// TwinCAT 3 PLC project PLC
// ProgramVersion: 3.1.4024.0
// libraries:
//   Tc2_Standard, * (Beckhoff Automation GmbH)
//   Tc2_System, * (Beckhoff Automation GmbH)
//   Tc3_Module, * (Beckhoff Automation GmbH)
//   VisuDialogs, * (System)
//   VisuSymbols,3.5.10.0,System
// project tree:
//   / GlobalTextList.TcGTLO (not stored), PlcTask.TcTTO, Visualization Manager.TcVMO (not stored)
//   POUs/ MAIN.TcPOU
//   VISUs/ Visualization.TcVIS
// real-time tasks:
//   TASK PlcTask: cycle T#10ms, priority 20, ADS port 350

CONFIGURATION PLC
    RESOURCE PLC ON TwinCAT3
        TASK PlcTask(INTERVAL := T#10ms, PRIORITY := 20);
        PROGRAM MAIN WITH PlcTask : MAIN;
    END_RESOURCE
END_CONFIGURATION

// ---- POUs/MAIN.TcPOU
PROGRAM MAIN
VAR
	bStartMotor : BOOL := FALSE;
	bStopMotor  : BOOL := FALSE;
	bServoMotor : BOOL;
	sr_MotorSetReset : SR;
END_VAR


sr_MotorSetReset(SET1:= bStartMotor,
				 RESET:= bStopMotor,
				 Q1 => bServoMotor);

END_PROGRAM

// ---- VISUs/Visualization.TcVIS
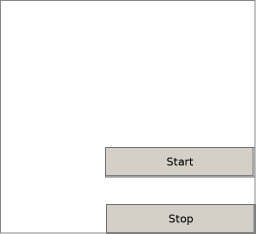
VISUALIZATION Visualization  // 256x234
    Button (105,147 150x30), "Start"
        OnMouseDown: execute { MAIN.bStartMotor := TRUE; }
        OnMouseUp: execute { MAIN.bStartMotor :=  FALSE; }
    Button (106,204 150x30), "Stop", pressed state: MAIN.bStopMotor
        OnMouseDown: execute { MAIN.bStopMotor := TRUE; }
        OnMouseUp: execute { MAIN.bStopMotor := FALSE; }
END_VISUALIZATION
